(* Logix 5000 project; controller cal1615 1756-L62 rev 20.19; software revision 20.05; part 56 of 82 *)
(* tags used below, declared in another part *)
   p23r17 : routine;
   p23r17_request_line_run : BOOL;
   FAULT : BOOL;   // Fault AFI
   p01r09_pb_global_reset : BOOL;   // System Modes PB: Global Fault Reset
   p01r13_line_running : BOOL;   // System Line Start Sequence Line Running
   p01r13_line_slow_ramp : BOOL;   // System Line Start Sequence Start Line to Slow Speed
   p01r13_permissive_drives : BOOL;   // System Line Start Sequence Permissive Drives
   p01r13_state : DINT;   // System Line Start Sequence Sequencer Step
   p23_ao_selected_speed : REAL;   // Impreg Metering Roll VFD Selected Speed
   p23_di_metering_roll : acs800_di_normal;   // Impreg Digital Inputs Metering Roll VFD
   p23_di_spring : acs800_di_normal;
   p23_do_Spring : acs800_do_normal;
   p23_param_min_start_tension : REAL;
   p23_param_mtr_jog_speed : REAL;   // System Parameter Metering Roll Jog Speed
   p23r09_mode_run : BOOL;   // Impreg Modes Pick Up Roll Run Mode
   p23r15_request_jog_fwd : BOOL;   // Impreg Metering Roll VFD Request Jog FWD
   p23r15_request_jog_rev : BOOL;   // Impreg Metering Roll VFD Request Jog REV
   p23r15_request_line_run : BOOL;   // Impreg Metering Roll VFD Request Line Run
   p23r17_adjusted_speed : REAL;
   p23r17_di_brake : BOOL;
   p23r17_di_therm : BOOL;
   p23r17_permissive_jog : BOOL;
   p23r17_permissive_run : BOOL;
   p23r17_request_jog_fwd : BOOL;
   p23r17_request_thread_fwd : BOOL;
   p23r17_request_thread_rev : BOOL;
   p23r17_selected_speed : REAL;
   p23r17_spd_adj : REAL;
   p23r17_sprng_assist_hmi_auto : BOOL;
   p23r17_sprng_assist_hmi_jog : BOOL;
   p23r17_timer_fault : TIMER[10];
   p23r17_timer_warning : TIMER[5];
   p23r17_zero_speed : BOOL;
   p24_di_edge_guide_auto : BOOL;   // Edge Control Inputs SS: Edge Guide Manual/Auto Auto
   p24_di_edge_guide_center : BOOL;   // Edge Control Inputs PB: Edge Guide Center
   p24_di_edge_guide_left : BOOL;   // Edge Control Inputs PB: Edge Guide Left
   p24_di_edge_guide_right : BOOL;   // Edge Control Inputs PB: Edge Guide Right
   p24_dint_to_hmi : DINT[16];
   p24r01 : routine;
   p24r02 : routine;   // Edge Control Misc Control
   p24r02_fault_exists : BOOL;
   p24r02_timer_fault : TIMER[4];   // Edge Control Misc Control Fault Delay
   p24r02_timer_warning : TIMER[4];   // Edge Control Misc Control Warning Delay
   p24r02_unack_fault : BOOL;   // Tension Stand 2 Misc Control Unacknowledged Fault Exists
   p24r02_unack_warning : BOOL;   // Tension Stand 2 Misc Control Unacknowledged Warning Exists
   p24r02_warning_exists : BOOL;
   p24r03 : routine;   // Edge Control Inputs
   p24r03_timer_fault : TIMER[4];   // Edge Control Inputs Fault Delay
   p24r03_timer_warning : TIMER[4];   // Edge Control Inputs Warning Delay
   p24r04 : routine;   // Edge Control Outputs
   p24r05 : routine;   // Edge Control Dint to HMI
   p24r06 : routine;   // Edge Control Real to HMI
   p24r07 : routine;   // Edge Control Alarms
   p24r08 : routine;   // Edge Control Warings
   p24r09 : routine;   // Tension Stand 2 Modes
   p24r10 : routine;   // Edge Control Edge Guide
   p25_ai_ts2_lc : REAL;   // System Metering Roll VFD Minimum Start Tension
   p25r11_request_thread_fwd : BOOL;   // Tension Stand 2 VFD Request Thread FWD
   p25r11_request_thread_rev : BOOL;   // Tension Stand 2 VFD Request Thread REV
   spring_spd_adj_prcnt : REAL;
(* P23_Impreg, continued *)

ROUTINE R17_SPRING_ASSIST_VFD   (* ladder *)
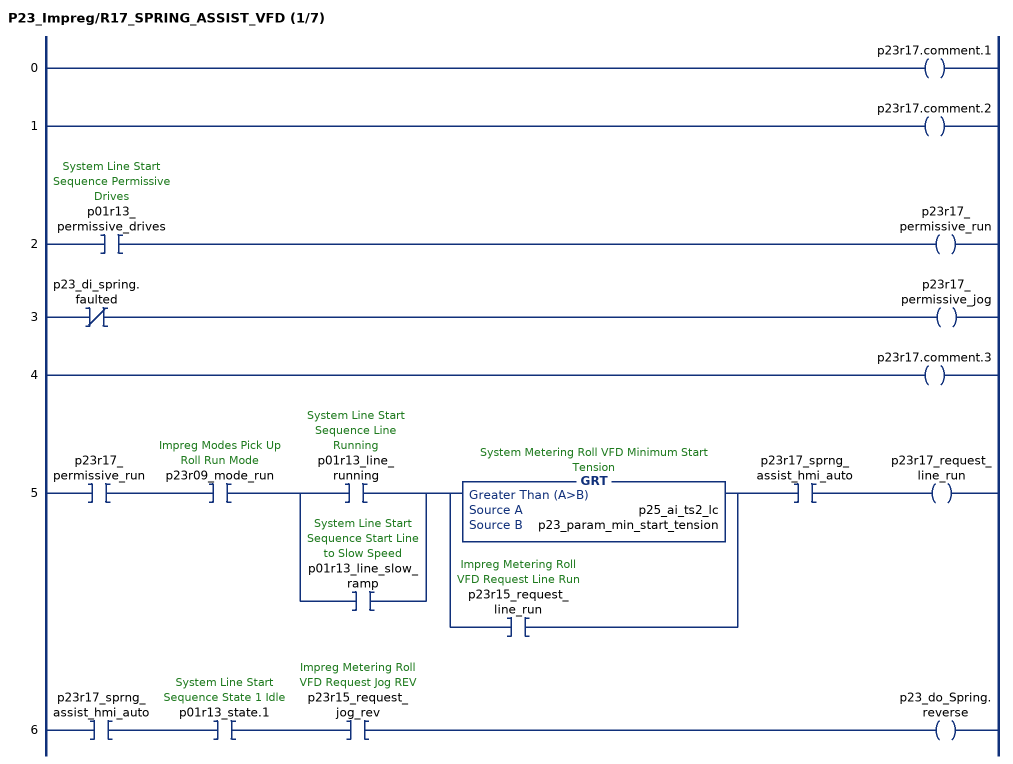
   0: OTE(p23r17.comment.1);
   1: OTE(p23r17.comment.2);
   2: XIC(p01r13_permissive_drives)OTE(p23r17_permissive_run);
   3: XIO(p23_di_spring.faulted)OTE(p23r17_permissive_jog);
   4: OTE(p23r17.comment.3);
   5: XIC(p23r17_permissive_run)XIC(p23r09_mode_run)[XIC(p01r13_line_running) ,XIC(p01r13_line_slow_ramp) ][GRT(p25_ai_ts2_lc,p23_param_min_start_tension) ,XIC(p23r15_request_line_run) ]XIC(p23r17_sprng_assist_hmi_auto)OTE(p23r17_request_line_run);
   6: XIC(p23r17_sprng_assist_hmi_auto)XIC(p01r13_state.1)XIC(p23r15_request_jog_rev)OTE(p23_do_Spring.reverse);
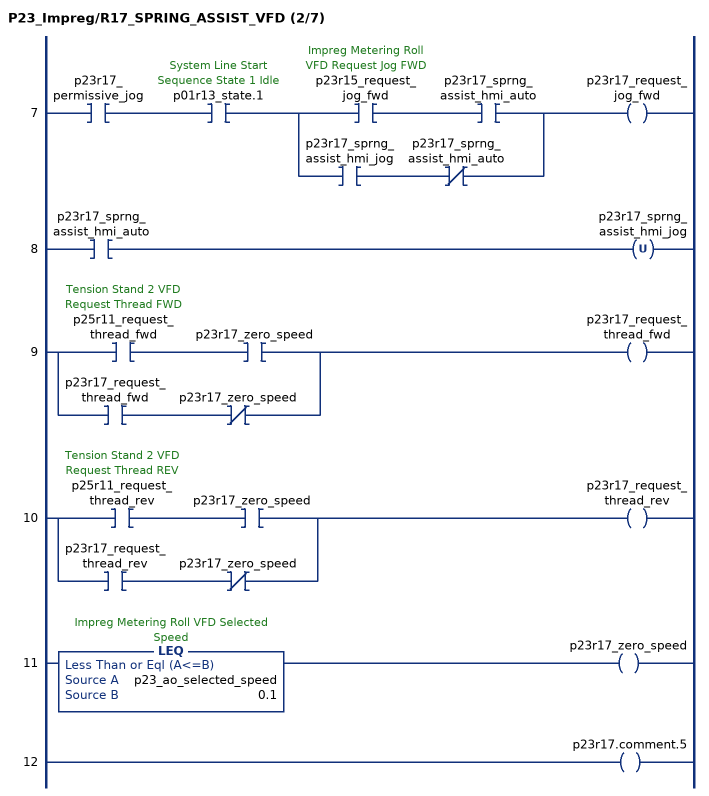
   7: XIC(p23r17_permissive_jog)XIC(p01r13_state.1)[XIC(p23r15_request_jog_fwd) XIC(p23r17_sprng_assist_hmi_auto) ,XIC(p23r17_sprng_assist_hmi_jog) XIO(p23r17_sprng_assist_hmi_auto) ]OTE(p23r17_request_jog_fwd);
   8: XIC(p23r17_sprng_assist_hmi_auto)OTU(p23r17_sprng_assist_hmi_jog);
   9: [XIC(p25r11_request_thread_fwd) XIC(p23r17_zero_speed) ,XIC(p23r17_request_thread_fwd) XIO(p23r17_zero_speed) ]OTE(p23r17_request_thread_fwd);
   10: [XIC(p25r11_request_thread_rev) XIC(p23r17_zero_speed) ,XIC(p23r17_request_thread_rev) XIO(p23r17_zero_speed) ]OTE(p23r17_request_thread_rev);
   11: LEQ(p23_ao_selected_speed,0.1)OTE(p23r17_zero_speed);
   12: OTE(p23r17.comment.5);
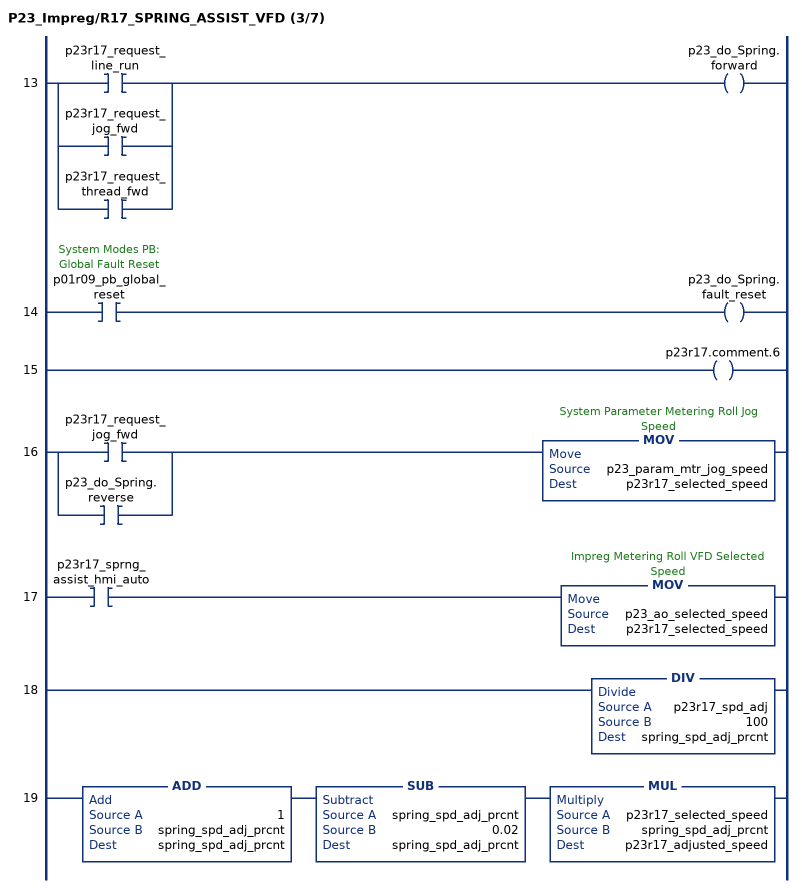
   13: [XIC(p23r17_request_line_run) ,XIC(p23r17_request_jog_fwd) ,XIC(p23r17_request_thread_fwd) ]OTE(p23_do_Spring.forward);
   14: XIC(p01r09_pb_global_reset)OTE(p23_do_Spring.fault_reset);
   15: OTE(p23r17.comment.6);
   16: [XIC(p23r17_request_jog_fwd) ,XIC(p23_do_Spring.reverse) ]MOV(p23_param_mtr_jog_speed,p23r17_selected_speed);
   17: XIC(p23r17_sprng_assist_hmi_auto)MOV(p23_ao_selected_speed,p23r17_selected_speed);
   18: DIV(p23r17_spd_adj,100,spring_spd_adj_prcnt);
   19: ADD(1,spring_spd_adj_prcnt,spring_spd_adj_prcnt)SUB(spring_spd_adj_prcnt,0.02,spring_spd_adj_prcnt)MUL(p23r17_selected_speed,spring_spd_adj_prcnt,p23r17_adjusted_speed);
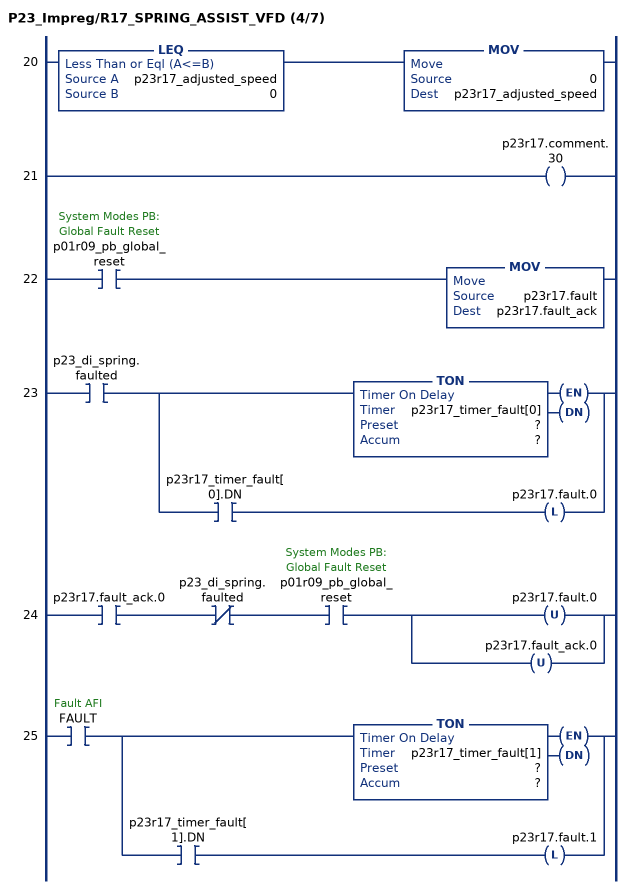
   20: LEQ(p23r17_adjusted_speed,0)MOV(0,p23r17_adjusted_speed);
   21: OTE(p23r17.comment.30);
   22: XIC(p01r09_pb_global_reset)MOV(p23r17.fault,p23r17.fault_ack);
   23: XIC(p23_di_spring.faulted)[TON(p23r17_timer_fault[0],?,?) ,XIC(p23r17_timer_fault[0].DN) OTL(p23r17.fault.0) ];
   24: XIC(p23r17.fault_ack.0)XIO(p23_di_spring.faulted)XIC(p01r09_pb_global_reset)[OTU(p23r17.fault.0) ,OTU(p23r17.fault_ack.0) ];
   25: XIC(FAULT)[TON(p23r17_timer_fault[1],?,?) ,XIC(p23r17_timer_fault[1].DN) OTL(p23r17.fault.1) ];
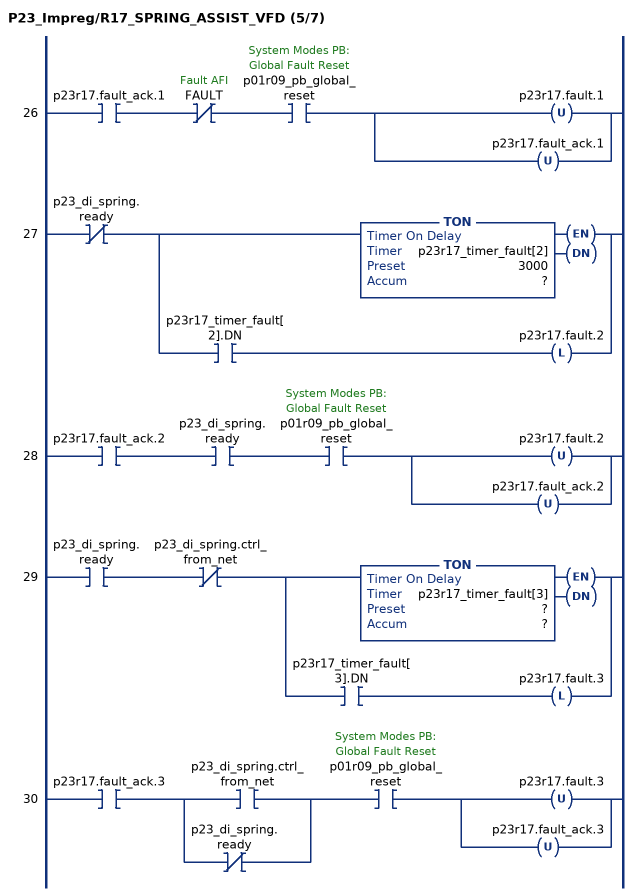
   26: XIC(p23r17.fault_ack.1)XIO(FAULT)XIC(p01r09_pb_global_reset)[OTU(p23r17.fault.1) ,OTU(p23r17.fault_ack.1) ];
   27: XIO(p23_di_spring.ready)[TON(p23r17_timer_fault[2],?,?) ,XIC(p23r17_timer_fault[2].DN) OTL(p23r17.fault.2) ];
   28: XIC(p23r17.fault_ack.2)XIC(p23_di_spring.ready)XIC(p01r09_pb_global_reset)[OTU(p23r17.fault.2) ,OTU(p23r17.fault_ack.2) ];
   29: XIC(p23_di_spring.ready)XIO(p23_di_spring.ctrl_from_net)[TON(p23r17_timer_fault[3],?,?) ,XIC(p23r17_timer_fault[3].DN) OTL(p23r17.fault.3) ];
   30: XIC(p23r17.fault_ack.3)[XIC(p23_di_spring.ctrl_from_net) ,XIO(p23_di_spring.ready) ]XIC(p01r09_pb_global_reset)[OTU(p23r17.fault.3) ,OTU(p23r17.fault_ack.3) ];
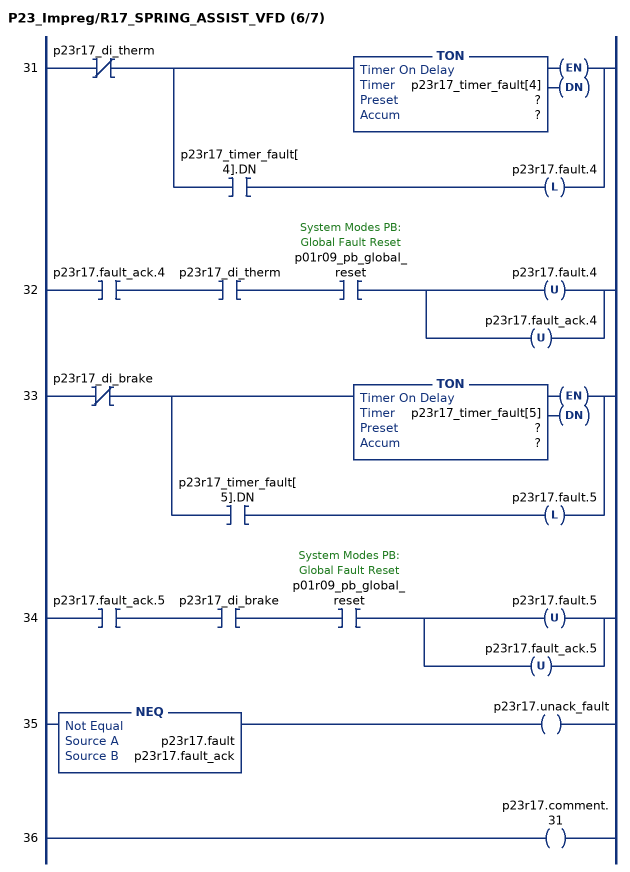
   31: XIO(p23r17_di_therm)[TON(p23r17_timer_fault[4],?,?) ,XIC(p23r17_timer_fault[4].DN) OTL(p23r17.fault.4) ];
   32: XIC(p23r17.fault_ack.4)XIC(p23r17_di_therm)XIC(p01r09_pb_global_reset)[OTU(p23r17.fault.4) ,OTU(p23r17.fault_ack.4) ];
   33: XIO(p23r17_di_brake)[TON(p23r17_timer_fault[5],?,?) ,XIC(p23r17_timer_fault[5].DN) OTL(p23r17.fault.5) ];
   34: XIC(p23r17.fault_ack.5)XIC(p23r17_di_brake)XIC(p01r09_pb_global_reset)[OTU(p23r17.fault.5) ,OTU(p23r17.fault_ack.5) ];
   35: NEQ(p23r17.fault,p23r17.fault_ack)OTE(p23r17.unack_fault);
   36: OTE(p23r17.comment.31);
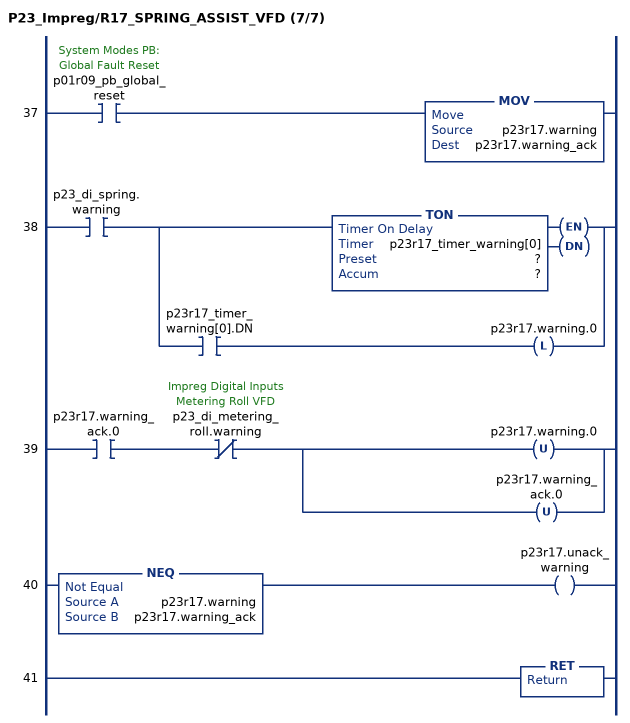
   37: XIC(p01r09_pb_global_reset)MOV(p23r17.warning,p23r17.warning_ack);
   38: XIC(p23_di_spring.warning)[TON(p23r17_timer_warning[0],?,?) ,XIC(p23r17_timer_warning[0].DN) OTL(p23r17.warning.0) ];
   39: XIC(p23r17.warning_ack.0)XIO(p23_di_metering_roll.warning)[OTU(p23r17.warning.0) ,OTU(p23r17.warning_ack.0) ];
   40: NEQ(p23r17.warning,p23r17.warning_ack)OTE(p23r17.unack_warning);
   41: RET();
END_ROUTINE
END_PROGRAM

PROGRAM P24_Edge_Control   (* main routine R01_Main *)

ROUTINE R01_Main   (* ladder *)
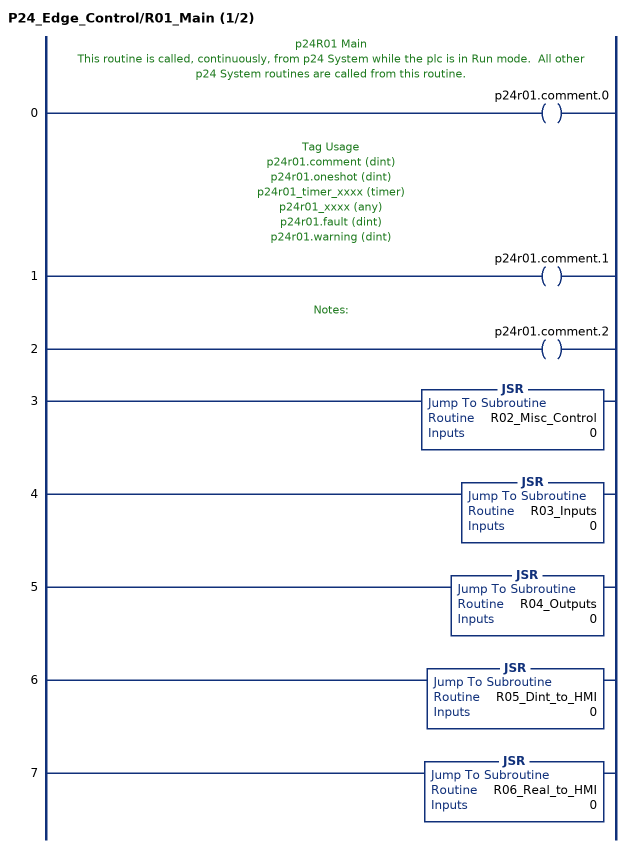
   // p24R01 Main
   // This routine is called, continuously, from p24 System while the plc is in Run mode.  All other p24 System routines are called from this routine.
   0: OTE(p24r01.comment.0);
   // Tag Usage
   // p24r01.comment (dint)
   // p24r01.oneshot (dint)
   // p24r01_timer_xxxx (timer)
   // p24r01_xxxx (any)
   // p24r01.fault (dint)
   // p24r01.warning (dint)
   1: OTE(p24r01.comment.1);
   // Notes:
   2: OTE(p24r01.comment.2);
   3: JSR(R02_Misc_Control,0);
   4: JSR(R03_Inputs,0);
   5: JSR(R04_Outputs,0);
   6: JSR(R05_Dint_to_HMI,0);
   7: JSR(R06_Real_to_HMI,0);
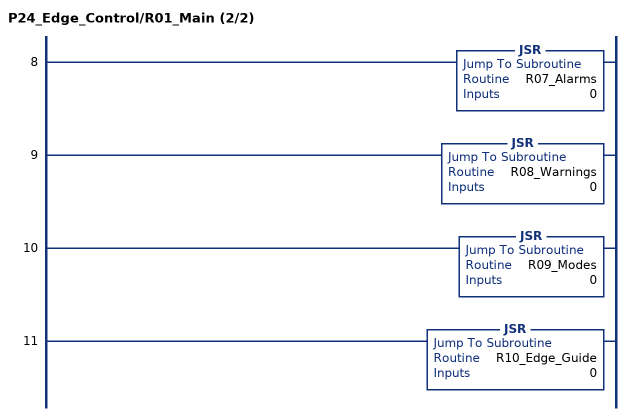
   8: JSR(R07_Alarms,0);
   9: JSR(R08_Warnings,0);
   10: JSR(R09_Modes,0);
   11: JSR(R10_Edge_Guide,0);
END_ROUTINE

ROUTINE R02_Misc_Control   (* ladder *)
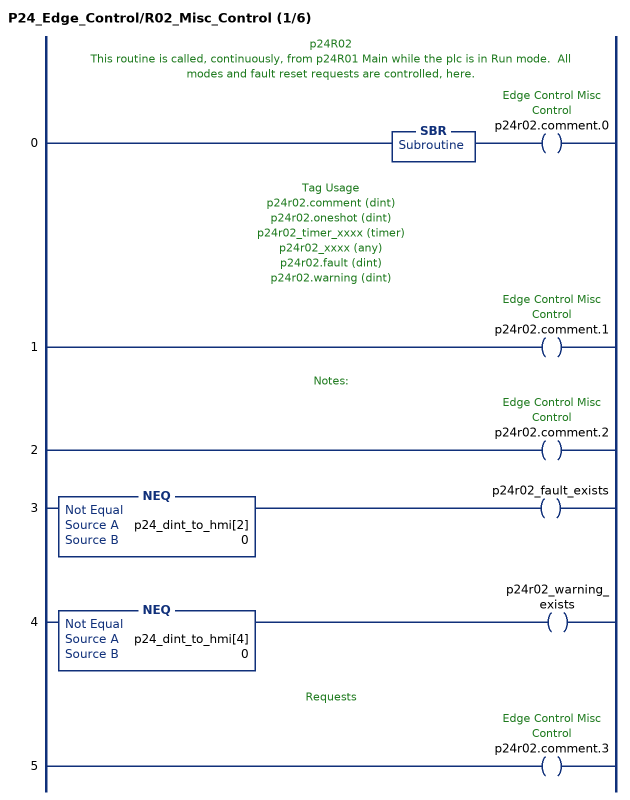
   // p24R02
   // This routine is called, continuously, from p24R01 Main while the plc is in Run mode.  All modes and fault reset requests are controlled, here.
   0: SBR()OTE(p24r02.comment.0);
   // Tag Usage
   // p24r02.comment (dint)
   // p24r02.oneshot (dint)
   // p24r02_timer_xxxx (timer)
   // p24r02_xxxx (any)
   // p24r02.fault (dint)
   // p24r02.warning (dint)
   1: OTE(p24r02.comment.1);
   // Notes:
   2: OTE(p24r02.comment.2);
   3: NEQ(p24_dint_to_hmi[2],0)OTE(p24r02_fault_exists);
   4: NEQ(p24_dint_to_hmi[4],0)OTE(p24r02_warning_exists);
   // Requests
   5: OTE(p24r02.comment.3);
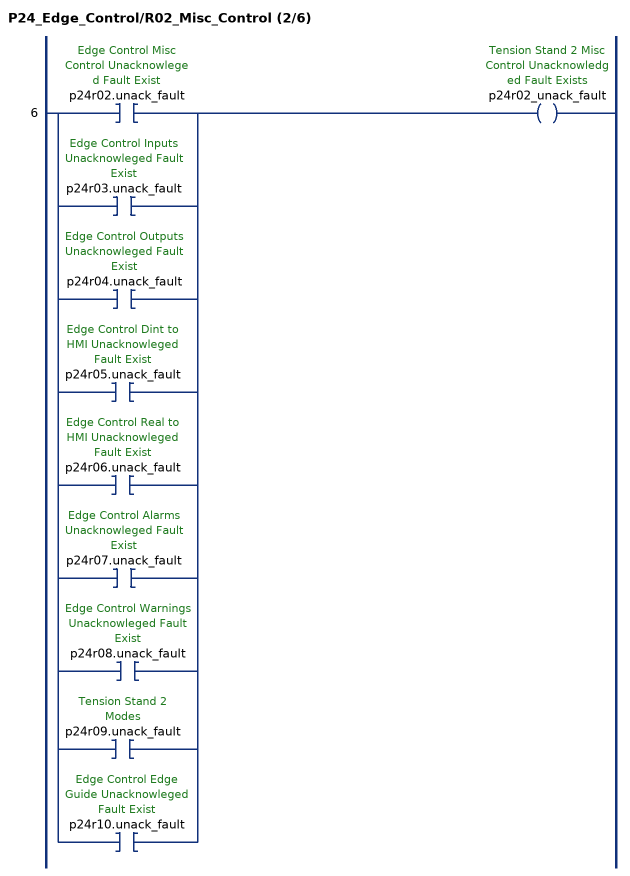
   6: [XIC(p24r02.unack_fault) ,XIC(p24r03.unack_fault) ,XIC(p24r04.unack_fault) ,XIC(p24r05.unack_fault) ,XIC(p24r06.unack_fault) ,XIC(p24r07.unack_fault) ,XIC(p24r08.unack_fault) ,XIC(p24r09.unack_fault) ,XIC(p24r10.unack_fault) ]OTE(p24r02_unack_fault);
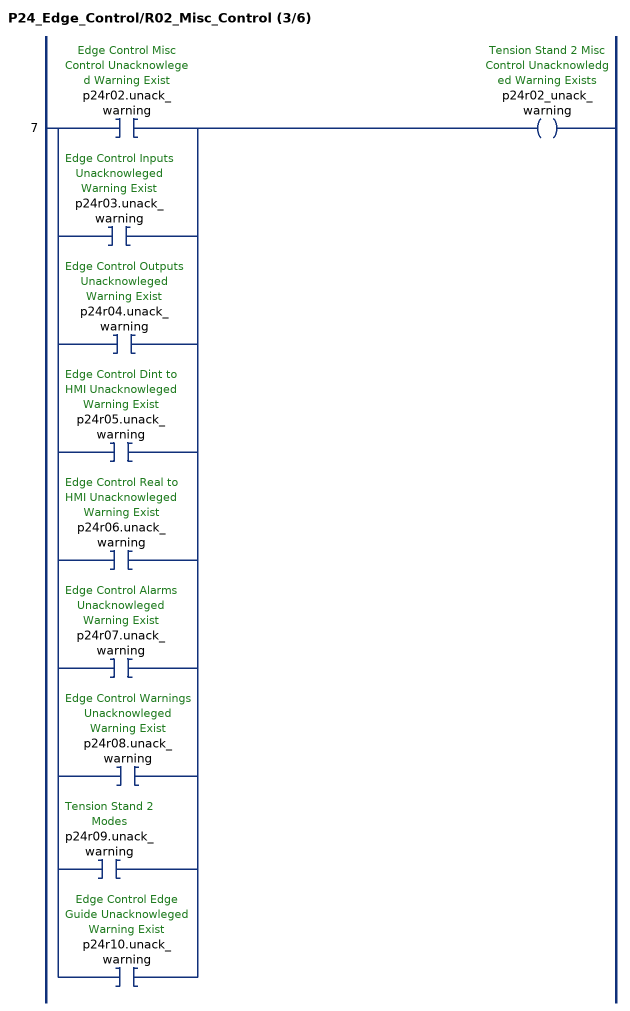
   7: [XIC(p24r02.unack_warning) ,XIC(p24r03.unack_warning) ,XIC(p24r04.unack_warning) ,XIC(p24r05.unack_warning) ,XIC(p24r06.unack_warning) ,XIC(p24r07.unack_warning) ,XIC(p24r08.unack_warning) ,XIC(p24r09.unack_warning) ,XIC(p24r10.unack_warning) ]OTE(p24r02_unack_warning);
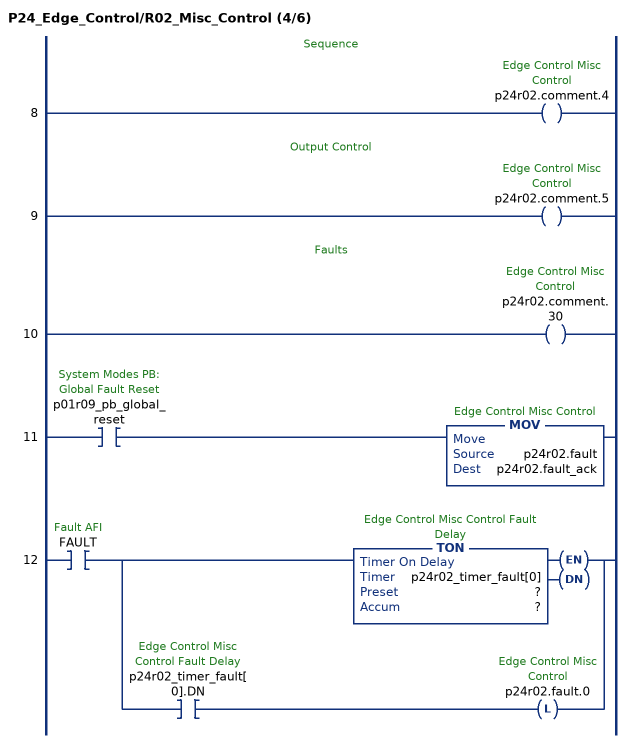
   // Sequence
   8: OTE(p24r02.comment.4);
   // Output Control
   9: OTE(p24r02.comment.5);
   // Faults
   10: OTE(p24r02.comment.30);
   11: XIC(p01r09_pb_global_reset)MOV(p24r02.fault,p24r02.fault_ack);
   12: XIC(FAULT)[TON(p24r02_timer_fault[0],?,?) ,XIC(p24r02_timer_fault[0].DN) OTL(p24r02.fault.0) ];
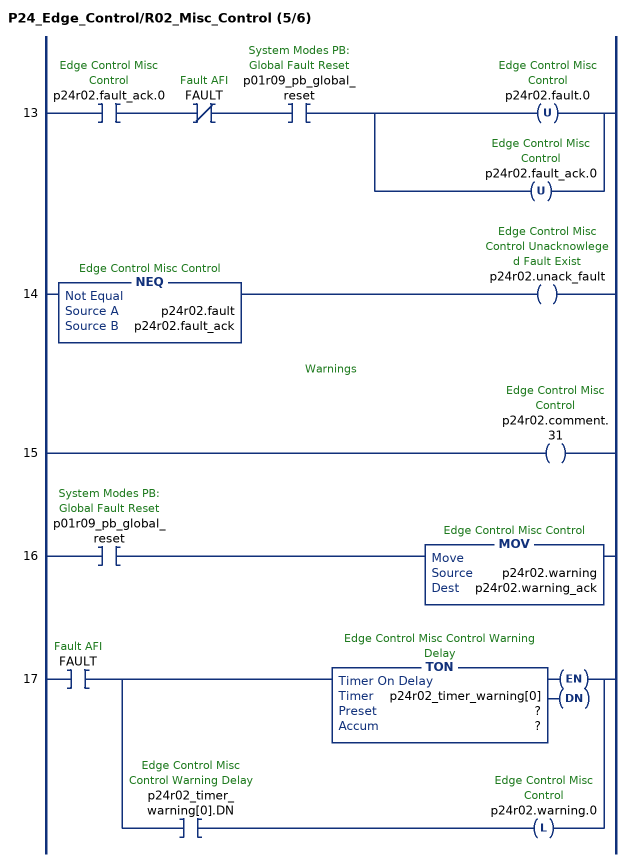
   13: XIC(p24r02.fault_ack.0)XIO(FAULT)XIC(p01r09_pb_global_reset)[OTU(p24r02.fault.0) ,OTU(p24r02.fault_ack.0) ];
   14: NEQ(p24r02.fault,p24r02.fault_ack)OTE(p24r02.unack_fault);
   // Warnings
   15: OTE(p24r02.comment.31);
   16: XIC(p01r09_pb_global_reset)MOV(p24r02.warning,p24r02.warning_ack);
   17: XIC(FAULT)[TON(p24r02_timer_warning[0],?,?) ,XIC(p24r02_timer_warning[0].DN) OTL(p24r02.warning.0) ];
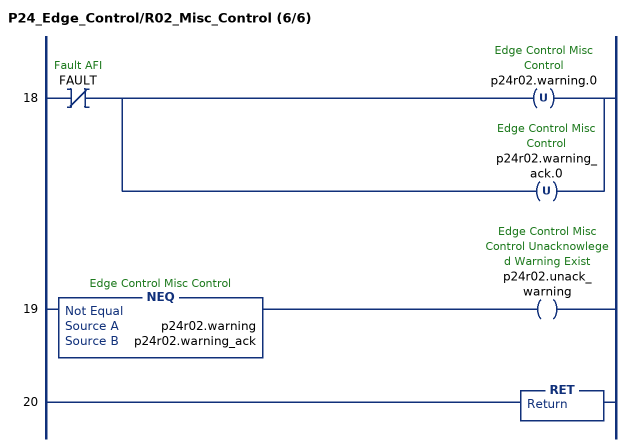
   18: XIO(FAULT)[OTU(p24r02.warning.0) ,OTU(p24r02.warning_ack.0) ];
   19: NEQ(p24r02.warning,p24r02.warning_ack)OTE(p24r02.unack_warning);
   20: RET();
END_ROUTINE

ROUTINE R03_Inputs   (* ladder *)
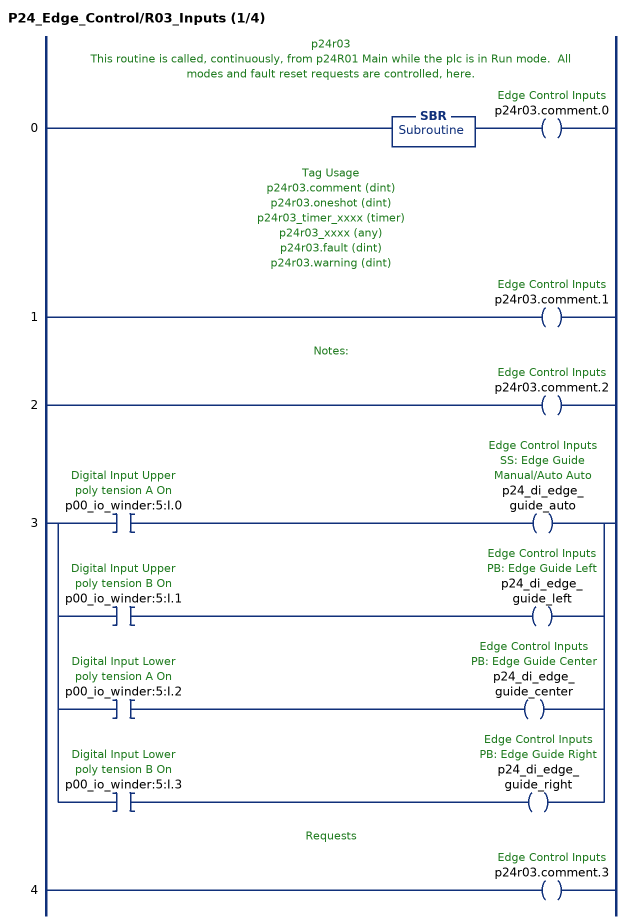
   // p24r03
   // This routine is called, continuously, from p24R01 Main while the plc is in Run mode.  All modes and fault reset requests are controlled, here.
   0: SBR()OTE(p24r03.comment.0);
   // Tag Usage
   // p24r03.comment (dint)
   // p24r03.oneshot (dint)
   // p24r03_timer_xxxx (timer)
   // p24r03_xxxx (any)
   // p24r03.fault (dint)
   // p24r03.warning (dint)
   1: OTE(p24r03.comment.1);
   // Notes:
   2: OTE(p24r03.comment.2);
   3: [XIC(p00_io_winder:5:I.0) OTE(p24_di_edge_guide_auto) ,XIC(p00_io_winder:5:I.1) OTE(p24_di_edge_guide_left) ,XIC(p00_io_winder:5:I.2) OTE(p24_di_edge_guide_center) ,XIC(p00_io_winder:5:I.3) OTE(p24_di_edge_guide_right) ];
   // Requests
   4: OTE(p24r03.comment.3);
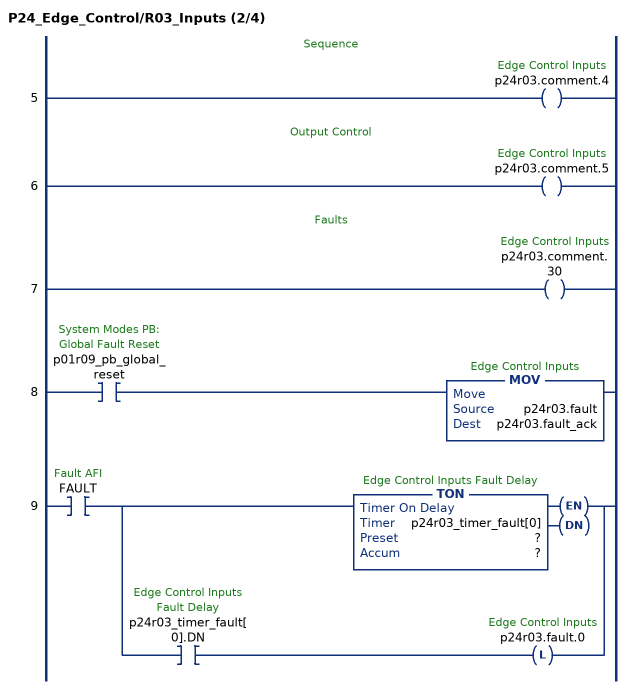
   // Sequence
   5: OTE(p24r03.comment.4);
   // Output Control
   6: OTE(p24r03.comment.5);
   // Faults
   7: OTE(p24r03.comment.30);
   8: XIC(p01r09_pb_global_reset)MOV(p24r03.fault,p24r03.fault_ack);
   9: XIC(FAULT)[TON(p24r03_timer_fault[0],?,?) ,XIC(p24r03_timer_fault[0].DN) OTL(p24r03.fault.0) ];
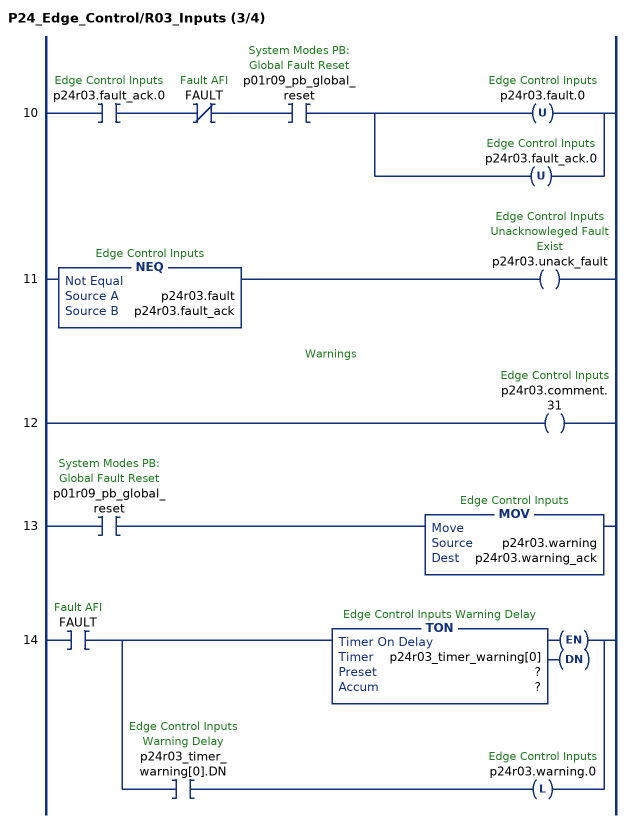
   10: XIC(p24r03.fault_ack.0)XIO(FAULT)XIC(p01r09_pb_global_reset)[OTU(p24r03.fault.0) ,OTU(p24r03.fault_ack.0) ];
   11: NEQ(p24r03.fault,p24r03.fault_ack)OTE(p24r03.unack_fault);
   // Warnings
   12: OTE(p24r03.comment.31);
   13: XIC(p01r09_pb_global_reset)MOV(p24r03.warning,p24r03.warning_ack);
   14: XIC(FAULT)[TON(p24r03_timer_warning[0],?,?) ,XIC(p24r03_timer_warning[0].DN) OTL(p24r03.warning.0) ];
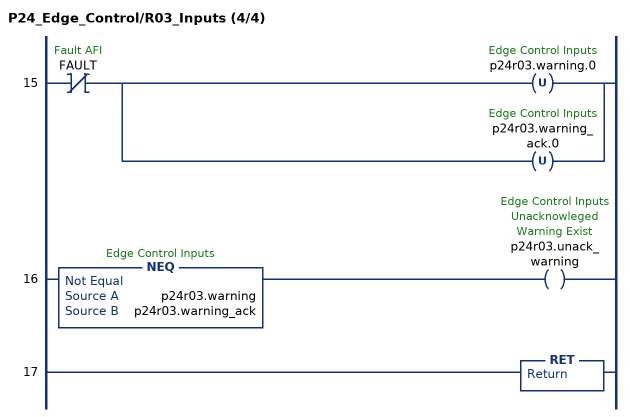
   15: XIO(FAULT)[OTU(p24r03.warning.0) ,OTU(p24r03.warning_ack.0) ];
   16: NEQ(p24r03.warning,p24r03.warning_ack)OTE(p24r03.unack_warning);
   17: RET();
END_ROUTINE
